FUNCTION_BLOCK Test_F_DateTimeAsString EXTENDS T_UnitTestBase
VAR
    TimeStruct : TIMESTRUCT := (wDay    := 23,
                                wMonth  := 12,
                                wYear   := 1945,
                                wHour   := 22,
                                wMinute := 20,
                                wSecond := 18);
END_VAR

METHOD Init
VAR_INPUT
END_VAR
END_METHOD

{attribute 'analysis' := '-33'} // inhibit unused variable warning
METHOD RunTest
AssertEquals_STRING(Expected := '22:20:18 23/12/1945',
                    Actual   := F_DateTimeAsString(TimeStruct),
                    Message  := 'F_DateTimeAsString(TimeStruct)');

TestCompleted := TRUE;
END_METHOD

END_FUNCTION_BLOCK

(* stored: Version 1.1.0.1, ProductVersion 3.1.4024.12
   POU Test_F_DateTimeAsString: Id {70721f54-ad56-0ed4-217d-cb50130dc051}, SpecialFunc None
   Method Init: Id {6952c4d8-351a-0e90-0fec-c54ed405976d}
   Method RunTest: Id {684b7a57-4fc7-02a8-1cd8-a5a40ff772fd} *)
